(* IEC 61131-3 sources: ATCMcontrol_Engineering/src/COM/softing/fc/AddOns/Softing/4CPCTarget/Libs/ATCM_Utility, 52 files *)

(* ---- BYTE_STRING_APPEND.st ---- *)
(*[[
    UserURL= "ATCM:BYTE_STRING_APPEND.htm"
]]*)

(* appends the byte string BSTR2 at the end of the byte string BSTR1 *)

FUNCTION BYTE_STRING_APPEND
VAR_IN_OUT
    BSTR1 : BYTE_STRING;
END_VAR
VAR_INPUT
    BSTR2 : BYTE_STRING;
END_VAR
VAR
    START_POS : DINT;
    COPY_LENGTH : DINT;
END_VAR

    COPY_LENGTH := BSTR2.SIZE;
    START_POS := BSTR1.SIZE;
    BSTR1.SIZE := START_POS+COPY_LENGTH;
    NATIVE
    	{
        	// appends the second bytestring to the first bytestring
    		int c;
            byte byteString1[],byteString2[];

            byteString1 = ((COM.softing.fc.CC.utility.ByteString)_bstr1).getByteString();
            byteString2 = ((COM.softing.fc.CC.utility.ByteString)_bstr2).getByteString();
    		for (c=0; c<_copy_length; c++) {
                byteString1[_start_pos+c] = byteString2[c];
            }
        }
    END_NATIVE;

END_FUNCTION

(* ---- BYTE_STRING_GET.ST ---- *)
(*[[
    UserURL= "ATCM:BYTE_STRING_GET.htm"
]]*)

FUNCTION BYTE_STRING_GET : BYTE
VAR_INPUT
    BSTR  : BYTE_STRING;
    INDEX : DINT;
END_VAR

inline{((COM.softing.fc.CC.utility.ByteString)%1).getByteAt(%2)}

END_FUNCTION

(* ---- BYTE_STRING_INIT.ST ---- *)
(*[[
    UserURL= "ATCM:BYTE_STRING_INIT.htm"
]]*)

(**
 * BYTE_STRING_INIT initializes the byte-string to the given value.
 * C-like \-quotes are supported to specify non-ascii characters.
 * example:
 * BYTE_STRING_INIT(bstr, "abc\x00\x01");
 *)

FUNCTION BYTE_STRING_INIT
VAR_IN_OUT
    BSTR  : BYTE_STRING;
END_VAR
VAR_INPUT
    VALUE : WSTRING; (* ASCII character string! *)
END_VAR
inline{((COM.softing.fc.CC.utility.ByteString)%1).initFromString(%2)}

END_FUNCTION

(* ---- BYTE_STRING_SET.ST ---- *)
(*[[
    UserURL= "ATCM:BYTE_STRING_SET.htm"
]]*)

FUNCTION BYTE_STRING_SET
VAR_IN_OUT
    BSTR  : BYTE_STRING;
END_VAR
VAR_INPUT
    INDEX : DINT;
    VALUE : BYTE;
END_VAR

inline{((COM.softing.fc.CC.utility.ByteString)%1).setByteAt(%2,%3)}

END_FUNCTION

(* ---- BYTE_STRING_SUBSTR.st ---- *)
(*[[
    UserURL= "ATCM:BYTE_STRING_SUBSTR.htm"
]]*)

(* extracts a sub- byte string from BSTR *)
(* the sub-string to be extracted is specified by a starting position POS *)
(* and a string length NUM *)

FUNCTION BYTE_STRING_SUBSTR
VAR_INPUT
    BSTR : BYTE_STRING;
    POS  : DINT;
    NUM  : DINT;
END_VAR
VAR_IN_OUT
    BSTR_SUB : BYTE_STRING;
END_VAR
VAR
    COPY_LENGTH : DINT;
END_VAR

    IF (POS < BSTR.SIZE) THEN
        IF (POS+NUM > BSTR.SIZE) THEN
            COPY_LENGTH := BSTR.SIZE-POS;
        ELSE
            COPY_LENGTH := NUM;
        END_IF;
    ELSE
        COPY_LENGTH := 0;
    END_IF;
    BSTR_SUB.SIZE := COPY_LENGTH;
    NATIVE
    	{
        	// extracts the given number of bytes at the given position from a bytestring
    		int c;
            byte sourceByteString[],subByteString[];
            sourceByteString = ((COM.softing.fc.CC.utility.ByteString)_bstr).getByteString();
            subByteString = ((COM.softing.fc.CC.utility.ByteString)_bstr_sub).getByteString();
    		for (c=0; c<_copy_length; c++) {
                subByteString[c] = sourceByteString[_pos+c];
            }
        }
    END_NATIVE;

END_FUNCTION

(* ---- BYTE_STRING_TO_WSTRING.ST ---- *)
(*[[
    UserURL= "ATCM:BYTE_STRING_TO_WSTRING.htm"
]]*)

(**
 * BYTE_STRING_TO_WSTRING converts a BYTE_STRING value into
 * human-readable form.
 * non-ascii characters will be escaped like "\xDD"
 *)

FUNCTION BYTE_STRING_TO_WSTRING : WSTRING
VAR_INPUT
    BSTR  : BYTE_STRING;
END_VAR

inline{%1.toString()}

END_FUNCTION

(* ---- BYTE_SWAP_DWORD.st ---- *)
(*[[
    UserURL= "ATCM:BYTE_SWAP_DWORD.htm"
]]*)

(* swaps from big to little endian byte order and vice versa *)

FUNCTION BYTE_SWAP_DWORD : DWORD
VAR_INPUT
    VALUE : DWORD;
END_VAR

    (* dummy assignment to avoid no return walue warnings *)
    BYTE_SWAP_DWORD := 0;
    NATIVE
        _byte_swap_dword =
            ((_value&(0xff<<0))<<24)|
            ((_value&(0xff<<8))<<8)|
            ((_value&(0xff<<16))>>>8)|
            ((_value&(0xff<<24))>>>24);
    END_NATIVE;

END_FUNCTION

(* ---- BYTE_SWAP_LWORD.st ---- *)
(*[[
    UserURL= "ATCM:BYTE_SWAP_LWORD.htm"
]]*)

(* swaps from big to little endian byte order and vice versa *)

FUNCTION BYTE_SWAP_LWORD:LWORD
VAR_INPUT
    VALUE : LWORD;
END_VAR

    (* dummy assignment to avoid no return walue warnings *)
    BYTE_SWAP_LWORD := 0;
    NATIVE
        _byte_swap_lword =
            ((_value&(0xffL<<0))<<56)|
            ((_value&(0xffL<<8))<<40)|
            ((_value&(0xffL<<16))<<24)|
            ((_value&(0xffL<<24))<<8)|
            ((_value&(0xffL<<32))>>>8)|
            ((_value&(0xffL<<40))>>>24)|
            ((_value&(0xffL<<48))>>>40)|
            ((_value&(0xffL<<56))>>>56);
    END_NATIVE;

END_FUNCTION

(* ---- BYTE_SWAP_WORD.st ---- *)
(*[[
    UserURL= "ATCM:BYTE_SWAP_WORD.htm"
]]*)

(* swaps from big to little endian byte order and vice versa *)

FUNCTION BYTE_SWAP_WORD : WORD
VAR_INPUT
    VALUE : WORD;
END_VAR

    (* dummy assignment to avoid no return walue warnings *)
    BYTE_SWAP_WORD := 0;
    NATIVE
        _byte_swap_word =
            ((_value&(0xff<<0))<<8)|
            ((_value&(0xff<<8))>>>8);
    END_NATIVE;

END_FUNCTION

(* ---- COPY_BOOL_FROM_BYTE_STRING.st ---- *)
(*[[
    UserURL= "ATCM:COPY_BOOL_FROM_BYTE_STRING.htm"
]]*)

(* returns a value copied from the byte string BSTR at the position POS *)

FUNCTION COPY_BOOL_FROM_BYTE_STRING : BOOL
VAR_IN_OUT
    POS : DINT;
    BSTR : BYTE_STRING;
END_VAR

    COPY_BOOL_FROM_BYTE_STRING :=
        LWORD_TO_BOOL(COPY_NUMERIC_FROM_BYTE_STRING(1,POS,BSTR));

END_FUNCTION

(* ---- COPY_BOOL_TO_BYTE_STRING.st ---- *)
(*[[
    UserURL= "ATCM:COPY_BOOL_TO_BYTE_STRING.htm"
]]*)

(* copies the value VALUE to the byte string BSTR at the position POS *)

FUNCTION COPY_BOOL_TO_BYTE_STRING
VAR_INPUT
    VALUE : BOOL;
END_VAR
VAR_IN_OUT
    POS : DINT;
    BSTR : BYTE_STRING;
END_VAR

    COPY_NUMERIC_TO_BYTE_STRING(BOOL_TO_LWORD(VALUE),1,POS,BSTR);

END_FUNCTION

(* ---- COPY_BYTE_FROM_BYTE_STRING.st ---- *)
(*[[
    UserURL= "ATCM:COPY_BYTE_FROM_BYTE_STRING.htm"
]]*)

(* returns a value copied from the byte string BSTR at the position POS *)

FUNCTION COPY_BYTE_FROM_BYTE_STRING : BYTE
VAR_IN_OUT
    POS : DINT;
    BSTR : BYTE_STRING;
END_VAR

    COPY_BYTE_FROM_BYTE_STRING := LWORD_TO_BYTE(
        COPY_NUMERIC_FROM_BYTE_STRING(1,POS,BSTR));

END_FUNCTION

(* ---- COPY_BYTE_TO_BYTE_STRING.st ---- *)
(*[[
    UserURL= "ATCM:COPY_BYTE_TO_BYTE_STRING.htm"
]]*)

(* copies the value VALUE to the byte string BSTR at the position POS *)

FUNCTION COPY_BYTE_TO_BYTE_STRING
VAR_INPUT
    VALUE : BYTE;
END_VAR
VAR_IN_OUT
    POS : DINT;
    BSTR : BYTE_STRING;
END_VAR

    COPY_NUMERIC_TO_BYTE_STRING(BYTE_TO_LWORD(VALUE),1,POS,BSTR);

END_FUNCTION

(* ---- COPY_DATE_FROM_BYTE_STRING.st ---- *)
(*[[
    UserURL= "ATCM:COPY_DATE_FROM_BYTE_STRING.htm"
]]*)

(* returns a value copied from the byte string BSTR at the position POS *)

FUNCTION COPY_DATE_FROM_BYTE_STRING : DATE
VAR_IN_OUT
    POS : DINT;
    BSTR : BYTE_STRING;
END_VAR
VAR
    LWORD_VALUE : LWORD;
END_VAR

    (* dummy assignment to avoid warnings, true value is assigned within native code *)
    COPY_DATE_FROM_BYTE_STRING := DATE#0001-01-01;
    LWORD_VALUE := COPY_NUMERIC_FROM_BYTE_STRING(4,POS,BSTR);

    NATIVE
        _copy_date_from_byte_string = (int) _lword_value;
    END_NATIVE;

END_FUNCTION

(* ---- COPY_DATE_TO_BYTE_STRING.st ---- *)
(*[[
    UserURL= "ATCM:COPY_DATE_TO_BYTE_STRING.htm"
]]*)

(* copies the value VALUE to the byte string BSTR at the position POS *)

FUNCTION COPY_DATE_TO_BYTE_STRING
VAR_INPUT
    VALUE : DATE;
END_VAR
VAR_IN_OUT
    POS : DINT;
    BSTR : BYTE_STRING;
END_VAR
VAR
    LWORD_VALUE : LWORD;
END_VAR

    NATIVE
        _lword_value = _value;
    END_NATIVE;

    COPY_NUMERIC_TO_BYTE_STRING(LWORD_VALUE,4,POS,BSTR);

END_FUNCTION

(* ---- COPY_DINT_FROM_BYTE_STRING.st ---- *)
(*[[
    UserURL= "ATCM:COPY_DINT_FROM_BYTE_STRING.htm"
]]*)

(* returns a value copied from the byte string BSTR at the position POS *)

FUNCTION COPY_DINT_FROM_BYTE_STRING : DINT
VAR_IN_OUT
    POS : DINT;
    BSTR : BYTE_STRING;
END_VAR

    COPY_DINT_FROM_BYTE_STRING :=
        LWORD_TO_DINT(COPY_NUMERIC_FROM_BYTE_STRING(4,POS,BSTR));

END_FUNCTION

(* ---- COPY_DINT_TO_BYTE_STRING.st ---- *)
(*[[
    UserURL= "ATCM:COPY_DINT_TO_BYTE_STRING.htm"
]]*)

(* copies the value VALUE to the byte string BSTR at the position POS *)

FUNCTION COPY_DINT_TO_BYTE_STRING
VAR_INPUT
    VALUE : DINT;
END_VAR
VAR_IN_OUT
    POS : DINT;
    BSTR : BYTE_STRING;
END_VAR

    COPY_NUMERIC_TO_BYTE_STRING(DINT_TO_LWORD(VALUE),4,POS,BSTR);

END_FUNCTION

(* ---- COPY_DT_FROM_BYTE_STRING.st ---- *)
(*[[
    UserURL= "ATCM:COPY_DT_FROM_BYTE_STRING.htm"
]]*)

(* returns a value copied from the byte string BSTR at the position POS *)

FUNCTION COPY_DT_FROM_BYTE_STRING : DATE_AND_TIME
VAR_IN_OUT
    POS : DINT;
    BSTR : BYTE_STRING;
END_VAR
VAR
    LWORD_VALUE : LWORD;
END_VAR

    (* dummy assignment to avoid warnings, true value is assigned within native code *)
    COPY_DT_FROM_BYTE_STRING := DATE_AND_TIME#0001-01-01-00:00:00.000;
    LWORD_VALUE := COPY_NUMERIC_FROM_BYTE_STRING(8,POS,BSTR);

    NATIVE
        _copy_dt_from_byte_string = _lword_value;
    END_NATIVE;

END_FUNCTION

(* ---- COPY_DT_TO_BYTE_STRING.st ---- *)
(*[[
    UserURL= "ATCM:COPY_DT_TO_BYTE_STRING.htm"
]]*)

(* copies the value VALUE to the byte string BSTR at the position POS *)

FUNCTION COPY_DT_TO_BYTE_STRING
VAR_INPUT
    VALUE : DATE_AND_TIME;
END_VAR
VAR_IN_OUT
    POS : DINT;
    BSTR : BYTE_STRING;
END_VAR
VAR
    LWORD_VALUE : LWORD;
END_VAR

    NATIVE
        _lword_value = _value;
    END_NATIVE;

    COPY_NUMERIC_TO_BYTE_STRING(LWORD_VALUE,8,POS,BSTR);

END_FUNCTION

(* ---- COPY_DWORD_FROM_BYTE_STRING.st ---- *)
(*[[
    UserURL= "ATCM:COPY_DWORD_FROM_BYTE_STRING.htm"
]]*)

(* returns a value copied from the byte string BSTR at the position POS *)

FUNCTION COPY_DWORD_FROM_BYTE_STRING : DWORD
VAR_IN_OUT
    POS : DINT;
    BSTR : BYTE_STRING;
END_VAR

    COPY_DWORD_FROM_BYTE_STRING := LWORD_TO_DWORD(
        COPY_NUMERIC_FROM_BYTE_STRING(4,POS,BSTR));

END_FUNCTION

(* ---- COPY_DWORD_TO_BYTE_STRING.st ---- *)
(*[[
    UserURL= "ATCM:COPY_DWORD_TO_BYTE_STRING.htm"
]]*)

(* copies the value VALUE to the byte string BSTR at the position POS *)

FUNCTION COPY_DWORD_TO_BYTE_STRING
VAR_INPUT
    VALUE : DWORD;
END_VAR
VAR_IN_OUT
    POS : DINT;
    BSTR : BYTE_STRING;
END_VAR

    COPY_NUMERIC_TO_BYTE_STRING(DWORD_TO_LWORD(VALUE),4,POS,BSTR);

END_FUNCTION

(* ---- COPY_LINT_FROM_BYTE_STRING.st ---- *)
(*[[
    UserURL= "ATCM:COPY_LINT_FROM_BYTE_STRING.htm"
]]*)

(* returns a value copied from the byte string BSTR at the position POS *)

FUNCTION COPY_LINT_FROM_BYTE_STRING : LINT
VAR_IN_OUT
    POS : DINT;
    BSTR : BYTE_STRING;
END_VAR

    COPY_LINT_FROM_BYTE_STRING :=
        LWORD_TO_LINT(COPY_NUMERIC_FROM_BYTE_STRING(8,POS,BSTR));

END_FUNCTION

(* ---- COPY_LINT_TO_BYTE_STRING.st ---- *)
(*[[
    UserURL= "ATCM:COPY_LINT_TO_BYTE_STRING.htm"
]]*)

(* copies the value VALUE to the byte string BSTR at the position POS *)

FUNCTION COPY_LINT_TO_BYTE_STRING
VAR_INPUT
    VALUE : LINT;
END_VAR
VAR_IN_OUT
    POS : DINT;
    BSTR : BYTE_STRING;
END_VAR

    COPY_NUMERIC_TO_BYTE_STRING(LINT_TO_LWORD(VALUE),8,POS,BSTR);

END_FUNCTION

(* ---- COPY_LREAL_FROM_BYTE_STRING.st ---- *)
(*[[
    UserURL= "ATCM:COPY_LREAL_FROM_BYTE_STRING.htm"
]]*)

(* returns a value copied from the byte string BSTR at the position POS *)

FUNCTION COPY_LREAL_FROM_BYTE_STRING : LREAL
VAR_IN_OUT
    POS : DINT;
    BSTR : BYTE_STRING;
END_VAR
VAR
    LWORD_VALUE : LWORD;
END_VAR

    (* dummy assignment to avoid warnings, true value is assigned within native code *)
    COPY_LREAL_FROM_BYTE_STRING := 0.0;
    LWORD_VALUE := COPY_NUMERIC_FROM_BYTE_STRING(8,POS,BSTR);

    NATIVE
        _copy_lreal_from_byte_string = Double.longBitsToDouble(_lword_value);
    END_NATIVE;

END_FUNCTION

(* ---- COPY_LREAL_TO_BYTE_STRING.st ---- *)
(*[[
    UserURL= "ATCM:COPY_LREAL_TO_BYTE_STRING.htm"
]]*)

(* copies the value VALUE to the byte string BSTR at the position POS *)

FUNCTION COPY_LREAL_TO_BYTE_STRING
VAR_INPUT
    VALUE : LREAL;
END_VAR
VAR_IN_OUT
    POS : DINT;
    BSTR : BYTE_STRING;
END_VAR
VAR
    LWORD_VALUE : LWORD;
END_VAR

    NATIVE
        _lword_value = Double.doubleToLongBits(_value);
    END_NATIVE;

    COPY_NUMERIC_TO_BYTE_STRING(LWORD_VALUE,8,POS,BSTR);

END_FUNCTION

(* ---- COPY_LWORD_FROM_BYTE_STRING.st ---- *)
(*[[
    UserURL= "ATCM:COPY_LWORD_FROM_BYTE_STRING.htm"
]]*)

(* returns a value copied from the byte string BSTR at the position POS *)

FUNCTION COPY_LWORD_FROM_BYTE_STRING : LWORD
VAR_IN_OUT
    POS : DINT;
    BSTR : BYTE_STRING;
END_VAR

    COPY_LWORD_FROM_BYTE_STRING := COPY_NUMERIC_FROM_BYTE_STRING(8,POS,BSTR);;

END_FUNCTION

(* ---- COPY_LWORD_TO_BYTE_STRING.st ---- *)
(*[[
    UserURL= "ATCM:COPY_LWORD_TO_BYTE_STRING.htm"
]]*)

(* copies the value VALUE to the byte string BSTR at the position POS *)

FUNCTION COPY_LWORD_TO_BYTE_STRING
VAR_INPUT
    VALUE : LWORD;
END_VAR
VAR_IN_OUT
    POS : DINT;
    BSTR : BYTE_STRING;
END_VAR

    COPY_NUMERIC_TO_BYTE_STRING(VALUE,8,POS,BSTR);

END_FUNCTION

(* ---- COPY_NUMERIC_FROM_BYTE_STRING.st ---- *)
(*[[
    UserURL= "ATCM:COPY_NUMERIC_FROM_BYTE_STRING.htm"
]]*)

(* returns a value copied from the byte string BSTR at the position POS *)
(* the width parameter specifies how many bytes will be used to extract the value *)

FUNCTION COPY_NUMERIC_FROM_BYTE_STRING : LWORD
VAR_INPUT
    WIDTH : DINT;
END_VAR
VAR_IN_OUT
    POS : DINT;
    BSTR : BYTE_STRING;
END_VAR

    COPY_NUMERIC_FROM_BYTE_STRING := 0;
    IF (BSTR.SIZE < POS+WIDTH) THEN
        POS := -1;
    ELSE
        NATIVE
        	{
            	// copies a given number of bytes from a bytestring
            	// the bytes to be read are all stored in the parameter value
            	// bytes are copied in big-endian order => most significant byte first
                int c;
                long result,unsignedByte;
                byte byteString[];

                byteString = ((COM.softing.fc.CC.utility.ByteString)_bstr).getByteString();
    			result = 0;
                for (c=0; c<_width; c++) {
        			unsignedByte = (long) byteString[_pos.getInt()+c];
    				result = (result<<8)|(unsignedByte&0xff);
        		}
    			_pos.putInt(_pos.getInt()+_width);
                _copy_numeric_from_byte_string = result;
        	}
        END_NATIVE;
    END_IF;

END_FUNCTION

(* ---- COPY_NUMERIC_TO_BYTE_STRING.st ---- *)
(*[[
    UserURL= "ATCM:COPY_NUMERIC_TO_BYTE_STRING.htm"
]]*)

(* copies the value VALUE to the byte string BSTR at the position POS *)
(* the width parameter specifies how many bytes will be used to store the value *)

FUNCTION COPY_NUMERIC_TO_BYTE_STRING
VAR_INPUT
    VALUE : LWORD;
    WIDTH : DINT;
END_VAR
VAR_IN_OUT
    POS : DINT;
    BSTR : BYTE_STRING;
END_VAR

    IF (BSTR.SIZE < POS+WIDTH) THEN
        BSTR.SIZE := POS+WIDTH;
    END_IF;
    NATIVE
    	{
        	// copies a given number of bytes to a bytestring
        	// the bytes to be stored are all contained in the value parameter
        	// bytes are copied in big-endian order => most significant byte first
    		int c,shiftDistance;
            byte byteValue,byteString[];

    		shiftDistance = 0;
            byteString = ((COM.softing.fc.CC.utility.ByteString)_bstr).getByteString();
    		for (c=0; c<_width; c++) {
    			byteString[_pos.getInt()+_width-(c+1)] =
                    (byte) ((_value&((0xffL)<<shiftDistance))>>>shiftDistance);
    			shiftDistance += 8;
    		}
   			_pos.putInt(_pos.getInt()+_width);
    	}
    END_NATIVE;

END_FUNCTION

(* ---- COPY_TIME_FROM_BYTE_STRING.st ---- *)
(*[[
    UserURL= "ATCM:COPY_TIME_FROM_BYTE_STRING.htm"
]]*)

(* returns a value copied from the byte string BSTR at the position POS *)

FUNCTION COPY_TIME_FROM_BYTE_STRING : TIME
VAR_IN_OUT
    POS : DINT;
    BSTR : BYTE_STRING;
END_VAR
VAR
    LWORD_VALUE : LWORD;
END_VAR

    (* dummy assignment to avoid warnings, true value is assigned within native code *)
    COPY_TIME_FROM_BYTE_STRING := TIME#0ms;
    LWORD_VALUE := COPY_NUMERIC_FROM_BYTE_STRING(8,POS,BSTR);

    NATIVE
        _copy_time_from_byte_string = _lword_value;
    END_NATIVE;

END_FUNCTION

(* ---- COPY_TIME_TO_BYTE_STRING.st ---- *)
(*[[
    UserURL= "ATCM:COPY_TIME_TO_BYTE_STRING.htm"
]]*)

(* copies the value VALUE to the byte string BSTR at the position POS *)

FUNCTION COPY_TIME_TO_BYTE_STRING
VAR_INPUT
    VALUE : TIME;
END_VAR
VAR_IN_OUT
    POS : DINT;
    BSTR : BYTE_STRING;
END_VAR
VAR
    LWORD_VALUE : LWORD;
END_VAR

    NATIVE
        _lword_value = _value;
    END_NATIVE;

    COPY_NUMERIC_TO_BYTE_STRING(LWORD_VALUE,8,POS,BSTR);

END_FUNCTION

(* ---- COPY_TOD_FROM_BYTE_STRING.st ---- *)
(*[[
    UserURL= "ATCM:COPY_TOD_FROM_BYTE_STRING.htm"
]]*)

(* returns a value copied from the byte string BSTR at the position POS *)

FUNCTION COPY_TOD_FROM_BYTE_STRING : TIME_OF_DAY
VAR_IN_OUT
    POS : DINT;
    BSTR : BYTE_STRING;
END_VAR
VAR
    LWORD_VALUE : LWORD;
END_VAR

    (* dummy assignment to avoid warnings, true value is assigned within native code *)
    COPY_TOD_FROM_BYTE_STRING := TIME_OF_DAY#00:00:00.000;
    LWORD_VALUE := COPY_NUMERIC_FROM_BYTE_STRING(4,POS,BSTR);

    NATIVE
        _copy_tod_from_byte_string = (int) _lword_value;
    END_NATIVE;

END_FUNCTION

(* ---- COPY_TOD_TO_BYTE_STRING.st ---- *)
(*[[
    UserURL= "ATCM:COPY_TOD_TO_BYTE_STRING.htm"
]]*)

(* copies the value VALUE to the byte string BSTR at the position POS *)

FUNCTION COPY_TOD_TO_BYTE_STRING
VAR_INPUT
    VALUE : TIME_OF_DAY;
END_VAR
VAR_IN_OUT
    POS : DINT;
    BSTR : BYTE_STRING;
END_VAR
VAR
    LWORD_VALUE : LWORD;
END_VAR

    NATIVE
        _lword_value = _value;
    END_NATIVE;

    COPY_NUMERIC_TO_BYTE_STRING(LWORD_VALUE,4,POS,BSTR);

END_FUNCTION

(* ---- COPY_WORD_FROM_BYTE_STRING.st ---- *)
(*[[
    UserURL= "ATCM:COPY_WORD_FROM_BYTE_STRING.htm"
]]*)

(* returns a value copied from the byte string BSTR at the position POS *)

FUNCTION COPY_WORD_FROM_BYTE_STRING : WORD
VAR_IN_OUT
    POS : DINT;
    BSTR : BYTE_STRING;
END_VAR

    COPY_WORD_FROM_BYTE_STRING := LWORD_TO_WORD(
        COPY_NUMERIC_FROM_BYTE_STRING(2,POS,BSTR));

END_FUNCTION

(* ---- COPY_WORD_TO_BYTE_STRING.st ---- *)
(*[[
    UserURL= "ATCM:COPY_WORD_TO_BYTE_STRING.htm"
]]*)

(* copies the value VALUE to the byte string BSTR at the position POS *)

FUNCTION COPY_WORD_TO_BYTE_STRING
VAR_INPUT
    VALUE : WORD;
END_VAR
VAR_IN_OUT
    POS : DINT;
    BSTR : BYTE_STRING;
END_VAR

    COPY_NUMERIC_TO_BYTE_STRING(WORD_TO_LWORD(VALUE),2,POS,BSTR);

END_FUNCTION

(* ---- COPY_WSTRING_FROM_BYTE_STRING.st ---- *)
(*[[
    UserURL= "ATCM:COPY_WSTRING_FROM_BYTE_STRING.htm"
]]*)

(* Returns a wstring copied from the byte string BSTR starting
 * at the position POS containing NUM bytes.
 * The NUM bytes are converted using the current codepage.
 *)
FUNCTION COPY_WSTRING_FROM_BYTE_STRING : WSTRING
VAR_INPUT
    NUM : DINT;
END_VAR
VAR_IN_OUT
    POS : DINT;
    BSTR : BYTE_STRING;
END_VAR

    COPY_WSTRING_FROM_BYTE_STRING := "";
    IF (BSTR.SIZE < POS+NUM) THEN
        POS := -1;
    ELSE
        NATIVE
            byte byteString[] = ((COM.softing.fc.CC.utility.ByteString)_bstr).getByteString();
            _copy_wstring_from_byte_string = new String(byteString, _pos.getInt(), _num);
            _pos.putInt(_pos.getInt()+_num);
        END_NATIVE;
    END_IF;

END_FUNCTION

(* ---- COPY_WSTRING_TO_BYTE_STRING.st ---- *)
(*[[
    UserURL= "ATCM:COPY_WSTRING_TO_BYTE_STRING.htm"
]]*)

(* Copies the value VALUE to the byte string BSTR starting at the position POS.
 * The unicode wstring VALUE will be converted to a multibyte representation
 * according to the current code page.
 * POS will be incremented by the actual number of multi bytes written to BSTR.
 *
 * Note: If a unicode char cannot be converted, the result is undefined.
 *)
FUNCTION COPY_WSTRING_TO_BYTE_STRING
VAR_INPUT
    VALUE : WSTRING;
END_VAR
VAR_IN_OUT
    POS : DINT;
    BSTR : BYTE_STRING;
END_VAR
VAR
    STRLEN : DINT;
END_VAR

native
    byte multibytes[] = _value.getBytes();
    _strlen = multibytes.length;
end_native;

    IF (BSTR.SIZE < POS+STRLEN) THEN
        BSTR.SIZE := POS+STRLEN;
    END_IF;

native
    byte byteString[] = ((COM.softing.fc.CC.utility.ByteString)_bstr).getByteString();
	int iStartPos = _pos.getInt();

    for(int c=0; c<_strlen; c++)
    {
        byteString[iStartPos+c] = multibytes[c];
	}
    _pos.putInt(iStartPos+_strlen);
END_NATIVE;

END_FUNCTION

(* ---- HI_BYTE.st ---- *)
(*[[
    UserURL= "ATCM:HI_BYTE.htm"
]]*)

(* extracts the high value BYTE from a WORD *)

FUNCTION HI_BYTE : BYTE
VAR_INPUT
    VALUE : WORD;
END_VAR
    (* dummy assignment to avoid no return walue warnings *)
    HI_BYTE := 0;
    NATIVE;
        _hi_byte = (_value&0xff00)>>>8;
    END_NATIVE;
END_FUNCTION

(* ---- HI_DWORD.st ---- *)
(*[[
    UserURL= "ATCM:HI_DWORD.htm"
]]*)

(* extracts the high value DWORD from a LWORD *)

FUNCTION HI_DWORD : DWORD
VAR_INPUT
    VALUE : LWORD;
END_VAR
    (* dummy assignment to avoid no return walue warnings *)
    HI_DWORD := 0;
    NATIVE;
        _hi_dword = (int) ((_value&0xffffffff00000000L)>>>32);
    END_NATIVE;
END_FUNCTION

(* ---- HI_WORD.st ---- *)
(*[[
    UserURL= "ATCM:HI_WORD.htm"
]]*)

(* extracts the high value WORD from a DWORD *)

FUNCTION HI_WORD : WORD
VAR_INPUT
    VALUE : DWORD;
END_VAR
    (* dummy assignment to avoid no return walue warnings *)
    HI_WORD := 0;
    NATIVE;
        _hi_word = (_value&0xffff0000)>>>16;
    END_NATIVE;
END_FUNCTION

(* ---- LO_BYTE.st ---- *)
(*[[
    UserURL= "ATCM:LO_BYTE.htm"
]]*)

(* extracts the low value BYTE from a WORD *)

FUNCTION LO_BYTE : BYTE
VAR_INPUT
    VALUE : WORD;
END_VAR
    (* dummy assignment to avoid no return walue warnings *)
    LO_BYTE := 0;
    NATIVE;
        _lo_byte = _value&0xff;
    END_NATIVE;
END_FUNCTION

(* ---- LO_DWORD.st ---- *)
(*[[
    UserURL= "ATCM:LO_DWORD.htm"
]]*)

(* extracts the low value DWORD from a LWORD *)

FUNCTION LO_DWORD : DWORD
VAR_INPUT
    VALUE : LWORD;
END_VAR
    (* dummy assignment to avoid no return walue warnings *)
    LO_DWORD := 0;
    NATIVE;
        _lo_dword = (int) (_value&0xffffffffL);
    END_NATIVE;
END_FUNCTION

(* ---- LO_WORD.st ---- *)
(*[[
    UserURL= "ATCM:LO_WORD.htm"
]]*)

(* extracts the low value WORD from a DWORD *)

FUNCTION LO_WORD : WORD
VAR_INPUT
    VALUE : DWORD;
END_VAR
    (* dummy assignment to avoid no return walue warnings *)
    LO_WORD := 0;
    NATIVE;
        _lo_word = _value&0xffff;
    END_NATIVE;
END_FUNCTION

(* ---- MAKE_DWORD.st ---- *)
(*[[
    UserURL= "ATCM:MAKE_DWORD.htm"
]]*)

(* combines two WORDs to a DWORD *)

FUNCTION MAKE_DWORD : DWORD
VAR_INPUT
    LO_WORD : WORD;
    HI_WORD : WORD;
END_VAR
    (* dummy assignment to avoid no return walue warnings *)
    MAKE_DWORD := 0;
    NATIVE;
        _make_dword = (((int) _hi_word)<<16)|(0xffff&_lo_word);
    END_NATIVE;
END_FUNCTION

(* ---- MAKE_LWORD.st ---- *)
(*[[
    UserURL= "ATCM:MAKE_LWORD.htm"
]]*)

(* combines two DWORDs to a LWORD *)

FUNCTION MAKE_LWORD : LWORD
VAR_INPUT
    LO_DWORD : DWORD;
    HI_DWORD : DWORD;
END_VAR
    (* dummy assignment to avoid no return walue warnings *)
    MAKE_LWORD := 0;
    NATIVE;
        _make_lword = (((long) _hi_dword)<<32)|(0xffffffffL&_lo_dword);
    END_NATIVE;
END_FUNCTION

(* ---- MAKE_WORD.st ---- *)
(*[[
    UserURL= "ATCM:MAKE_WORD.htm"
]]*)

(* combines two BYTEs to a WORD *)

FUNCTION MAKE_WORD : WORD
VAR_INPUT
    LO_BYTE : BYTE;
    HI_BYTE : BYTE;
END_VAR
    (* dummy assignment to avoid no return walue warnings *)
    MAKE_WORD := 0;
    NATIVE;
        _make_word = (((short) _hi_byte)<<8)|(0xff&_lo_byte);
    END_NATIVE;
END_FUNCTION

(* ---- COPY_STRUCT_FROM_BYTE_STRING.st ---- *)
(* copies the data contained in the bytes string at the position POS to the structure STR *)
(* note that components with non-base types are ignored (arrays and structures) *)
(* string typed structure components are stored with a terminating zero-character *)
(* this is necessary to be able to restore a previously saved string from the byte string *)
FUNCTION_BLOCK COPY_STRUCT_FROM_BYTE_STRING
    VAR_IN_OUT
        STR : ANY_DERIVED;
        POS : DINT;
        BSTR : BYTE_STRING;
    END_VAR
    VAR
        BOOL_VAL : BOOL;
        LREAL_VAL : LREAL;
        DINT_VAL : DINT;
        LINT_VAL : LINT;
        WSTRING_VAL : WSTRING;
        WSTRING_LENGTH : DINT;
        BSTR_SIZE : DINT;
    END_VAR

    BSTR_SIZE := BSTR.SIZE;

    NATIVE
        {
            boolean stringEndPosFound;
        	int componentId,stringEndPos;
            byte byteString[];
        	FcObject componentObject;
            COM.softing.fc.CC.util.ObjectDirectoryEx stStruct;
        	ObjectDescriptor componentDescriptor,structureDescriptor;
        	java.util.Enumeration componentNameEnumerator;

            stStruct = (COM.softing.fc.CC.util.ObjectDirectoryEx) _str;
        	structureDescriptor = stStruct.getOD();
        	componentId = 0;
        	componentNameEnumerator = stStruct.getNameEnum();
            while (componentNameEnumerator.hasMoreElements() && (_pos.getInt() != -1)) {
                componentNameEnumerator.nextElement();
        		componentObject = stStruct.getObjectByID(componentId);
        		componentDescriptor = componentObject.getOD();
        		if(componentObject instanceof FcBool) {
    END_NATIVE;
                    BOOL_VAL := COPY_BOOL_FROM_BYTE_STRING(POS,BSTR);
    NATIVE
                    if (_pos.getInt() != -1) {
                        ((FcBool)componentObject).putBool(_bool_val.getBool());
                    }
            	} else if (componentObject instanceof FcDouble) {
    END_NATIVE;
                    LREAL_VAL := COPY_LREAL_FROM_BYTE_STRING(POS,BSTR);
    NATIVE
                    if (_pos.getInt() != -1) {
                        ((FcDouble)componentObject).putDouble(_lreal_val.getDouble());
                    }
           		} else if (componentObject instanceof FcInt) {
    END_NATIVE;
                    DINT_VAL := COPY_DINT_FROM_BYTE_STRING(POS,BSTR);
    NATIVE
                    if (_pos.getInt() != -1) {
                        ((FcInt)componentObject).putInt(_dint_val.getInt());
                    }
           		} else if (componentObject instanceof FcLong) {
    END_NATIVE;
                    LINT_VAL := COPY_LINT_FROM_BYTE_STRING(POS,BSTR);
    NATIVE
                    if (_pos.getInt() != -1) {
                        ((FcLong)componentObject).putLong(_lint_val.getLong());
                    }
           		} else if (componentObject instanceof FcString) {
                    byteString = ((COM.softing.fc.CC.commFB.ByteString)_bstr).getByteString();
                    stringEndPosFound = false;
                    stringEndPos = _pos.getInt();
                    while ((stringEndPos < _bstr_size.getInt()) && (! stringEndPosFound)) {
                        if (byteString[stringEndPos] == 0) {
                            stringEndPosFound = true;
                        } else {
                            stringEndPos++;
                        }
                    }
                    if (stringEndPosFound) {
                        _wstring_length.putInt(stringEndPos-_pos.getInt());
    END_NATIVE;
                        WSTRING_VAL := COPY_WSTRING_FROM_BYTE_STRING(WSTRING_LENGTH,POS,BSTR);
                        IF (POS <> -1) THEN
                            POS := POS+1;
                        END_IF;
    NATIVE
                    } else {
                        _pos.putInt(-1);
                    }
                    if (_pos.getInt() != -1) {
                        ((FcString)componentObject).putString(_wstring_val.getString());
                    }
           		}
           		componentId++;
           	}
        }
    END_NATIVE;
END_FUNCTION_BLOCK

(* ---- COPY_STRUCT_TO_BYTE_STRING.st ---- *)
(* copies the data contained in the structure STR to the byte string BSTR at the position POS *)
(* note that components with non-base types are ignored (arrays and structures) *)
(* string typed structure components are stored with a terminating zero-character *)
(* this is necessary to be able to restore a previously saved string from the byte string *)
FUNCTION_BLOCK COPY_STRUCT_TO_BYTE_STRING
    VAR_IN_OUT
        STR : ANY_DERIVED;
        POS : DINT;
        BSTR : BYTE_STRING;
    END_VAR
    VAR
        BOOL_VAL : BOOL;
        LREAL_VAL : LREAL;
        DINT_VAL : DINT;
        LINT_VAL : LINT;
        WSTRING_VAL : WSTRING;
    END_VAR
    NATIVE
        {
        	int componentId;
            COM.softing.fc.CC.util.ObjectDirectoryEx stStruct;
        	FcObject componentObject;
        	ObjectDescriptor componentDescriptor,structureDescriptor;
        	java.util.Enumeration componentNameEnumerator;

            stStruct = (COM.softing.fc.CC.util.ObjectDirectoryEx) _str;
        	structureDescriptor = stStruct.getOD();
        	componentId = 0;
        	componentNameEnumerator = stStruct.getNameEnum();
            while (componentNameEnumerator.hasMoreElements() && (_pos.getInt() != -1)) {
                componentNameEnumerator.nextElement();
        		componentObject = stStruct.getObjectByID(componentId);
        		componentDescriptor = componentObject.getOD();
        		if(componentObject instanceof FcBool) {
                    _bool_val.putBool(((FcBool)componentObject).getBool());
    END_NATIVE;
                    COPY_BOOL_TO_BYTE_STRING(BOOL_VAL,POS,BSTR);
    NATIVE
            	} else if (componentObject instanceof FcDouble) {
                    _lreal_val.putDouble(((FcDouble)componentObject).getDouble());
    END_NATIVE;
                    COPY_LREAL_TO_BYTE_STRING(LREAL_VAL,POS,BSTR);
    NATIVE
           		} else if (componentObject instanceof FcInt) {
                    _dint_val.putInt(((FcInt)componentObject).getInt());
    END_NATIVE;
                    COPY_DINT_TO_BYTE_STRING(DINT_VAL,POS,BSTR);
    NATIVE
           		} else if (componentObject instanceof FcLong) {
                    _lint_val.putLong(((FcLong)componentObject).getLong());
    END_NATIVE;
                    COPY_LINT_TO_BYTE_STRING(LINT_VAL,POS,BSTR);
    NATIVE
           		} else if (componentObject instanceof FcString) {
                    _wstring_val.putString(((FcString)componentObject).getString());
    END_NATIVE;
                    COPY_WSTRING_TO_BYTE_STRING(WSTRING_VAL,POS,BSTR);
                    IF (POS <> -1) THEN
                        COPY_BYTE_TO_BYTE_STRING(0,POS,BSTR);
                    END_IF;
    NATIVE
           		}
           		componentId++;
           	}
        }
    END_NATIVE;
END_FUNCTION_BLOCK

(* ---- RCV.ST ---- *)
(* Communication Function Blocks, see IEC 1131-5
 * Implements the RCV communication function block
 *
*)
FUNCTION_BLOCK RCV      (* Interlocked control, responder*)
VAR_INPUT
    EN_R   : BOOL;          (* Enable to receive data *)
    RESP   : BOOL (*R_EDGE*);   (* Request to send response data *)
    ID     : COMM_CHANNEL;  (* Communication channel *)
    R_ID   : WSTRING;       (* Remote function block *)
    EXPECT : DINT;          (* non-IEC: number of bytes to receive *)
(*    SD_1   : ANY;*)           (* User data to send *)
(*    SD_m   : ANY; *)
END_VAR

VAR_OUTPUT
NDR    : BOOL;              (* New user data received *)
ERROR  : BOOL;              (* New non-zero STATUS received *)
STATUS : DINT;              (* Last detected status *)

RD_1   : WSTRING; (*ANY*)       (* Received user data *)
(*RD_n   : ANY;*)         (*  It is not required that m=n *)
END_VAR(*  either m, n, or both may be 0*)

VAR_NATIVE#movetop
import COM.softing.fc.CC.commFB.*;
END_VAR

    (* is not implemented yet !! *)
    ERROR := TRUE;
    STATUS := CFB_ErrNotImpl;

NATIVE
END_NATIVE;

END_FUNCTION_BLOCK

(* ---- SEND.ST ---- *)
(* Communication Function Blocks, see IEC 1131-5
 * Implements the SEND communication function block
 *
*)
FUNCTION_BLOCK SEND     (* Interlocked control, requester*)
VAR_INPUT
    REQ    : BOOL (*R_EDGE*);       (* Request to send with raising edge*)
    R      : BOOL (*R_EDGE*);       (* Reset local, remote function *)
    ID     : COMM_CHANNEL;      (* Communication channel *)
    R_ID   : WSTRING;           (* Remote function block *)
    SD_1   : WSTRING;  (*ANY*)  (* User data to send *)
END_VAR

VAR_OUTPUT
    NDR    : BOOL;          (* New user data received *)
    ERROR  : BOOL;        (* New non-zero STATUS received *)
    STATUS : DINT;        (* Last detected status *)
(*    RD_1   : ANY;*)         (* Received user data *)
END_VAR                 (*   either m, n, or both may be 0*)
VAR_NATIVE#movetop
import COM.softing.fc.CC.commFB.*;
END_VAR

    (* is not implemented yet !! *)
    ERROR := TRUE;
    STATUS := CFB_ErrNotImpl;

NATIVE
END_NATIVE;

END_FUNCTION_BLOCK

(* ---- STATUS.ST ---- *)
(* Communication Function Blocks, see IEC 1131-5
 * Implements the STATUS communication function block
 *
*)
FUNCTION_BLOCK STATUS   (* Device verification - requester *)
VAR_INPUT
    REQ    : BOOL (*R_EDGE*);   (* Request *)
    ID     : COMM_CHANNEL;  (* Communication channel *)
END_VAR

VAR_OUTPUT
    NDR    : BOOL;        (* New user data received *)
    ERROR  : BOOL;        (* New non-zero STATUS received *)
    STATUS : DINT;        (* Last detected status *)
    PHYS   : DINT;        (* Physical status of remote *)
                          (*   communication partner   *)
    LOG    : DINT;        (* Logical status of remote *)
                          (*   communication partner   *)
    LOCAL  : ARRAY[0..7] OF WORD;  (* Local status of remote *)
END_VAR
VAR_NATIVE#movetop
import COM.softing.fc.CC.commFB.*;
END_VAR

    (* is not implemented yet !! *)
    ERROR := TRUE;
    STATUS := CFB_ErrNotImpl;
NATIVE
END_NATIVE;

END_FUNCTION_BLOCK

(* ---- USTATUS.ST ---- *)
(* Communication Function Blocks, see IEC 1131-5
 * Implements the USTATUS communication function block
 *
*)
FUNCTION_BLOCK USTATUS  (* Device verification - receiver *)
VAR_INPUT
    EN_R   : BOOL;        (* Enable to receive data *)
    ID     : COMM_CHANNEL;(* Communication channel *)
END_VAR

VAR_OUTPUT
    NDR    : BOOL;        (* New user data received *)
    ERROR  : BOOL;        (* New non-zero STATUS received *)
    STATUS : DINT;        (* Last detected status *)
    PHYS   : DINT;        (* Physical status of remote *)
                          (*   communication partner   *)
    LOG    : DINT;        (* Logical status of remote *)
                          (*   communication partner   *)
    LOCAL  : ARRAY[0..7] OF WORD; (* Local status of remote *)
                          (*   communication partner   *)
END_VAR
VAR_NATIVE#movetop
import COM.softing.fc.CC.commFB.*;
END_VAR

    (* is not implemented yet !! *)
    ERROR := TRUE;
    STATUS := CFB_ErrNotImpl;
NATIVE
END_NATIVE;

END_FUNCTION_BLOCK
